PROGRAM MAIN
VAR

END_VAR

Global.secImp := NOT(Global.secImp);

END_PROGRAM

(* stored: Version 1.1.0.1, ProductVersion 3.1.4024.13
   POU MAIN: Id {1ebefdd1-3e03-4aac-b0d7-9cb2e38b8084}, SpecialFunc None *)
